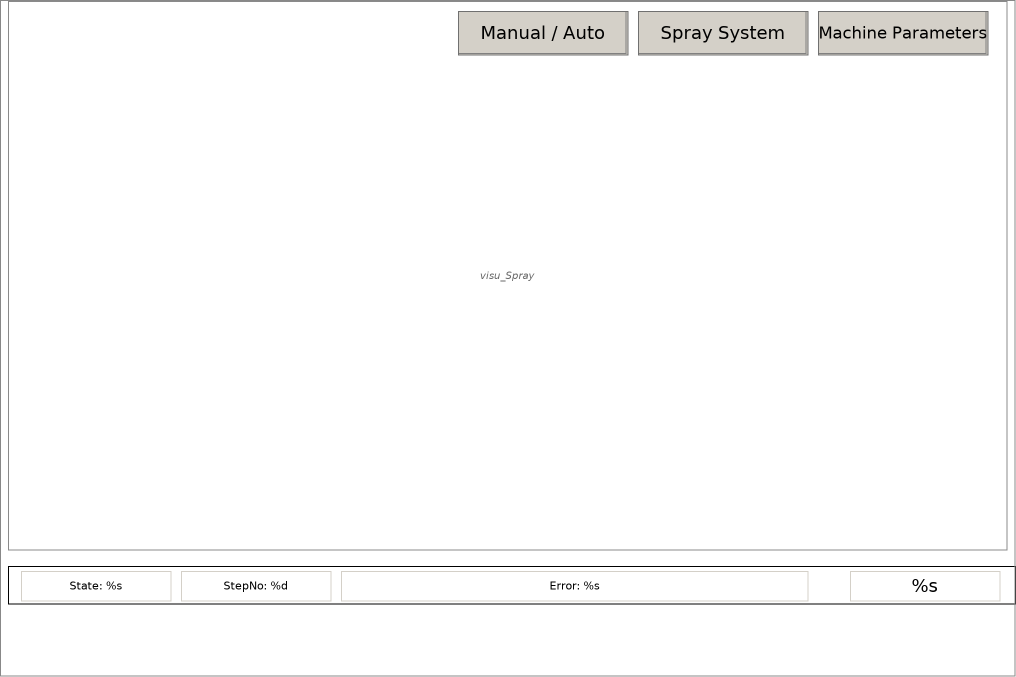
VISUALIZATION visu_Nav  // 1016x677
    Frame (8,1 999x549), frame switch variable: GVL_Nav.nPage
        shows visu_Spray()
        shows visu_Params()
    Button (638,11 170x44), "Spray System"
        p2175578022: SEL(GVL_Nav.abNavActive[0], 16#FF2D6FE0, 16#FF1FA34A)
        OnMouseClick: FrameSelectionChange Selection=SelectedFrame=ec7dd251-7f6b-4bd4-83c6-e8d232fe81a4, GlobSel=IndExpr=0, AssignType=Expression, SelType=Globally, SelectionStep=SelectedAction=SwitchNext
        OnMouseClick: execute { GVL_Nav.nPage := 0; }
    Button (818,11 170x44), "Machine Parameters"
        p2175578022: SEL(GVL_Nav.abNavActive[1], 16#FF2D6FE0, 16#FF1FA34A)
        OnMouseClick: FrameSelectionChange Selection=Selection=-1, GlobSel=IndExpr=1, AssignType=Expression, SelType=Globally, SelectionStep=SelectedAction=SwitchNext
        OnMouseClick: execute { GVL_Nav.nPage := 1; }
    Rectangle (8,566 1008x38)
    Textfield (21,571 150x30), "State: %s", text variable: PRG_Spray.sStateText
    Textfield (181,571 150x30), "StepNo: %d", text variable: TO_INT(MAIN.eState)
    Textfield (341,571 467x30), "Error: %s", text variable: PRG_Spray.sErrorText
    Textfield (850,571 150x30), "%s", text variable: PRG_Spray.sModeText
        p55702900: PRG_Spray.cModeColor
    Button (458,11 170x44), "Manual / Auto"
        p2175578022: PRG_Spray.cModeColor
        OnMouseClick: toggle PRG_Spray.bCmdAuto
    Line (956,676)
END_VISUALIZATION

(* stored: Version 1.1.0.1, ProductVersion 3.1.4026.18
   Visu visu_Nav: Id {2526f0b0-6f88-4b99-aca3-e87290d6c39d} *)
